// TIA Portal V20 export
DATA_BLOCK "DB_ChillerTermotek"   // DB540
// stored: AutoNumber false, InstanceOfName FB_ChillerTermotek, InstanceOfType FB
"FB_ChillerTermotek"
   // VAR
   //    sTimeHeadChillerHighPressure { S7_SetPoint := 'True'} : TON_TIME;
   //    sTimeHeadChillerWaterTemperature { S7_SetPoint := 'True'} : TON_TIME;
   //    sTimeHeadChillerAmbiantTemperature { S7_SetPoint := 'True'} : TON_TIME;
   //    sTimeOutFlowHeadChiller : TON_TIME;
   //    sTimeOutLevelHeadChiller { S7_SetPoint := 'True'} : TON_TIME;
   //    sTimeOutHeadChillerGood : TON_TIME;
   //    sTimeSourceChillerHighPressure { S7_SetPoint := 'True'} : TON_TIME;
   //    sTimeSourceChillerWaterTemperature { S7_SetPoint := 'True'} : TON_TIME;
   //    sTimeSourceChillerAmbiantTemperature { S7_SetPoint := 'True'} : TON_TIME;
   //    sTimeOutFlowSourceChiller : TON_TIME;
   //    sTimeOutLevelSourceChiller { S7_SetPoint := 'True'} : TON_TIME;
   //    sTimeOutSourceChillerGood : TON_TIME;
   // END_VAR
BEGIN
END_DATA_BLOCK
